FUNCTION_BLOCK eIXconfig (* Service Interface Function Block Type *)
  (* Standard: 61499-2; Description: Copyright (c) 2025 Maximilian Scharf This program and the accompanying materials are made available under the terms of the Eclipse Public License 2.0 which is available at https://www.eclipse.org/legal/epl-2.0/ SPDX-License-Identifier: EPL-2.0 *)
  (* Version 3.0, 2025-04-14, Franz Höpfinger, HR Agrartechnik GmbH, Made Version 3.0.0 inspired by Work from Patrick Aigner *)
  (* Version 1.0, 2025-05-05, Maximilian Scharf *)
  PACKAGE eclipse4diac::io::eio;
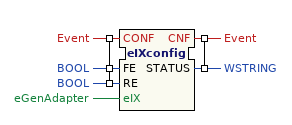
  EVENT_INPUT
    CONF WITH FE, RE; (* Configure Request *)
  END_EVENT
  EVENT_OUTPUT
    CNF WITH STATUS; (* Confirmation of Requested Service *)
  END_EVENT
  VAR_INPUT
    FE : BOOL; (* Falling Edge Trigger Enable *)
    RE : BOOL; (* Rising Edge Trigger Enable *)
  END_VAR
  VAR_OUTPUT
    STATUS : WSTRING; (* Service Status *)
  END_VAR
  SOCKETS
    eIX : eclipse4diac::io::eio::eGenAdapter; (* Connection to eIO Instance *)
  END_SOCKETS
END_FUNCTION_BLOCK
